PROGRAM Alarming
VAR
	bInit 		: BOOL := TRUE;
	bSendMsg	: BOOL;
	fbMsg		: FB_TcMessage;
END_VAR

IF bInit THEN
	bInit := FALSE;
	fbMsg.CreateEx(TC_Events.MyEventClass.MyMessage, 0);
END_IF

IF bSendMsg THEN
	bSendMsg := FALSE;
	fbMsg.Send(0);
END_IF

END_PROGRAM

(* stored: Version 1.1.0.1, ProductVersion 3.1.4024.12
   POU Alarming: Id {ecf07fd6-f111-49f0-9642-0a1d64acee76}, SpecialFunc None *)
